SUBAPPLICATION Vorsteuerventil_2B (* Subapplication Type *)
  (* Standard: 61499-2 *)
  (* Version 1.0, 2023-01-29, Franz *)
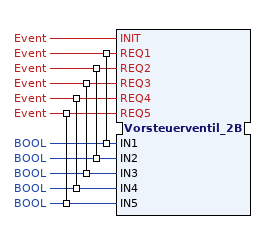
  EVENT_INPUT
    INIT;
    REQ1 WITH IN1;
    REQ2 WITH IN2;
    REQ3 WITH IN3;
    REQ4 WITH IN4;
    REQ5 WITH IN5;
  END_EVENT
  VAR_INPUT
    IN1 : BOOL;
    IN2 : BOOL;
    IN3 : BOOL;
    IN4 : BOOL;
    IN5 : BOOL;
  END_VAR
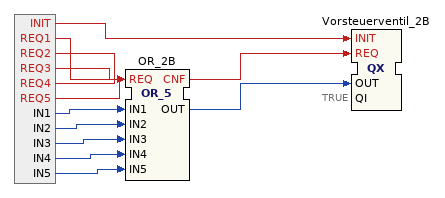
  FBS
    OR_2B : OR_5;
    Vorsteuerventil_2B : QX(QI := TRUE);
  END_FBS
  EVENT_CONNECTIONS
    REQ1 TO OR_2B.REQ;
    REQ2 TO OR_2B.REQ;
    REQ3 TO OR_2B.REQ;
    REQ4 TO OR_2B.REQ;
    REQ5 TO OR_2B.REQ;
    INIT TO Vorsteuerventil_2B.INIT;
    OR_2B.CNF TO Vorsteuerventil_2B.REQ;
  END_CONNECTIONS
  DATA_CONNECTIONS
    IN1 TO OR_2B.IN1;
    IN2 TO OR_2B.IN2;
    IN3 TO OR_2B.IN3;
    IN4 TO OR_2B.IN4;
    IN5 TO OR_2B.IN5;
    OR_2B.OUT TO Vorsteuerventil_2B.OUT;
  END_CONNECTIONS
END_SUBAPPLICATION
